TYPE DUT EXTENDS AXIS_REF :
STRUCT
END_STRUCT
END_TYPE

(* stored: Version 1.1.0.1
   DUT DUT: Id {067be2d9-b4ff-46eb-baad-abcefb8c1686} *)
